// TwinCAT 3 PLC project SmartHome_ReferenceLibrary
// Title: Smart Home Library
// Company: Oleksandr Tiutyk
// ProjectVersion: 0.0.0.1
// Description: OOP conceps demo for smart home
// ProgramVersion: 3.1.4026.20
// libraries:
//   Tc2_Standard, * (Beckhoff Automation GmbH)
//   Tc2_System, * (Beckhoff Automation GmbH)
// project tree:
//   Device/ DEVICE_STATE.TcDUT, IInputDevice.TcIO, IDevice.TcIO, IOutputDevice.TcIO
//   / SmartHome.TcPOU
// real-time tasks:
//   TASK PlcTask: cycle T#10ms, priority 20, ADS port 350
//   TASK PlcTask1: cycle T#10ms, priority 21, ADS port 351

// ---- Device/DEVICE_STATE.TcDUT
{attribute 'qualified_only'}
{attribute 'strict'}
{attribute 'to_string'}
TYPE DEVICE_STATE :
(
	FAULT := 0,
	WORKING
);
END_TYPE

// ---- Device/IInputDevice.TcIO
INTERFACE IInputDevice EXTENDS IDevice

METHOD ReadInputs
END_METHOD

END_INTERFACE

// ---- Device/IDevice.TcIO
INTERFACE IDevice EXTENDS __SYSTEM.IQueryInterface

{attribute 'monitoring' := 'call'}
PROPERTY Name : STRING
GET
END_GET
END_PROPERTY

{attribute 'monitoring' := 'call'}
PROPERTY Place : STRING
GET
END_GET
END_PROPERTY

{attribute 'monitoring' := 'call'}
PROPERTY State : DEVICE_STATE
GET
END_GET
END_PROPERTY

END_INTERFACE

// ---- Device/IOutputDevice.TcIO
INTERFACE IOutputDevice EXTENDS IDevice

METHOD WriteOutputs
END_METHOD

END_INTERFACE

// ---- SmartHome.TcPOU
FUNCTION_BLOCK ABSTRACT SmartHome
VAR_GENERIC CONSTANT
    _DeviceCount : UDINT := 1;
END_VAR
VAR_OUTPUT
	Devices : ARRAY [0.._DeviceCount - 1] OF IDevice;
END_VAR
VAR
	_SavedDeviceStates : ARRAY [0.._DeviceCount - 1] OF DEVICE_STATE;
	
	_LogMessageCounter : UDINT;
END_VAR

METHOD PUBLIC Execute
updateInputDevices();

OnTick();

updateOutputDevices();

saveDevicesState();
END_METHOD

//FB_Init is always available implicitly and it is used primarily for initialization.
//The return value is not evaluated. For a specific influence, you can also declare the
//methods explicitly and provide additional code there with the standard initialization
//code. You can evaluate the return value.
METHOD FB_Init: BOOL
VAR_INPUT
    bInitRetains: BOOL; // TRUE: the retain variables are initialized (reset warm / reset cold)
    bInCopyCode: BOOL;  // TRUE: the instance will be copied to the copy code afterward (online change)   
END_VAR
Devices := GetDeviceArray();
END_METHOD

METHOD PROTECTED ABSTRACT GetDeviceArray : ARRAY [0.._DeviceCount - 1] OF IDevice
END_METHOD

METHOD PRIVATE logDevicesState
VAR
	i : UDINT;
	message : STRING;
END_VAR
FOR i := 0 TO _DeviceCount - 1 DO
	IF Devices[i].State = DEVICE_STATE.FAULT AND_THEN _SavedDeviceStates[i] <> DEVICE_STATE.FAULT THEN
		_LogMessageCounter := _LogMessageCounter + 1;
		
		message := Tc2_Standard.CONCAT(
			Tc2_Standard.CONCAT(
				Tc2_Standard.CONCAT('#', TO_STRING(_LogMessageCounter)),
				Tc2_Standard.CONCAT(': ', 'Device "')
			),
			Tc2_Standard.CONCAT(
				Tc2_Standard.CONCAT(Devices[i].Name, '" at "'),
				Tc2_Standard.CONCAT(Devices[i].Place, '" is in fault state')
			)
		);
			
		Tc2_System.ADSLOGSTR(msgCtrlMask := Tc2_System.Global_Variables.ADSLOG_MSGTYPE_ERROR, message, '');
	ELSIF Devices[i].State = DEVICE_STATE.WORKING AND_THEN _SavedDeviceStates[i] <> DEVICE_STATE.WORKING THEN
		_LogMessageCounter := _LogMessageCounter + 1;

		message := Tc2_Standard.CONCAT(
			Tc2_Standard.CONCAT(
				Tc2_Standard.CONCAT('#', TO_STRING(_LogMessageCounter)),
				Tc2_Standard.CONCAT(': ', 'Device "')
			),
			Tc2_Standard.CONCAT(
				Tc2_Standard.CONCAT(Devices[i].Name, '" at "'),
				Tc2_Standard.CONCAT(Devices[i].Place, '" is in working state')
			)
		);
			
		Tc2_System.ADSLOGSTR(msgCtrlMask := Tc2_System.Global_Variables.ADSLOG_MSGTYPE_HINT, message, '');		
	END_IF
END_FOR
END_METHOD

METHOD PROTECTED OnTick
logDevicesState();
END_METHOD

METHOD PRIVATE saveDevicesState
VAR
	i : UDINT;
END_VAR
FOR i := 0 TO _DeviceCount - 1 DO
	_SavedDeviceStates[i] := Devices[i].State;
END_FOR
END_METHOD

METHOD PRIVATE updateInputDevices
VAR
	i : UDINT;
	device : IDevice;
	inputDevice : IInputDevice;
END_VAR
FOR i := 0 TO _DeviceCount - 1 DO
	device := Devices[i];
	
	IF __QUERYINTERFACE(device, inputDevice) THEN
		inputDevice.ReadInputs();		
	END_IF
END_FOR
END_METHOD

METHOD PRIVATE updateOutputDevices
VAR
	i : UDINT;
	device : IDevice;
	outputDevice : IOutputDevice;
END_VAR
FOR i := 0 TO _DeviceCount - 1 DO
	device := Devices[i];
	
	IF __QUERYINTERFACE(device, outputDevice) THEN
		outputDevice.WriteOutputs();		
	END_IF
END_FOR
END_METHOD

END_FUNCTION_BLOCK
